Staubli VAL3: J_MoveTo.pgx

program J_MoveTo(jointRx x_jPoint, tool x_tTool, mdesc x_mDesc, num x_nMoveType, bool& x_bReached)
  local bool l_bReached
  local joint l_jJoint
begin

    switch x_nMoveType
      case 0
        if pointToJoint(x_tTool,herej(),jointToPoint(x_tTool,world,x_jPoint),l_jJoint)
          movel(jointToPoint(x_tTool,world,x_jPoint),x_tTool,x_mDesc)
        else
          x_bReached=true
        endIf
      break
      case 1
        movej(x_jPoint,x_tTool,x_mDesc)
      break
    endSwitch

  end
